Yaskawa INFORM job: PARK-POS-ZONE-4-AUTO.JBI

/JOB
//NAME PARK-POS-ZONE-4-AUTO
//POS
///NPOS 1,1,0,0,0,0
///TOOL 0
///POSTYPE PULSE
///PULSE
C00000=75016,-48988,-40123,-68352,57928,88844
BC00000=79980
//INST
///DATE 2018/10/01 18:24
///ATTR SC,RW
///GROUP1 RB1,BS1
NOP
MOVJ C00000 BC00000 VJ=15.00
END
